//{attribute 'qualified_only'}
{attribute 'strict'}
TYPE E_MotionCommand :
(
	eNoCommand,
	ePower,
	eMoveAbsolute,
	eMoveRelative,
	eMoveVelocity,
	eHalt,
	eGearIn,
	eGearOut
);
END_TYPE

(* stored: Version 1.1.0.1, ProductVersion 3.1.4024.12
   DUT E_MotionCommand: Id {1ca8bf13-8b28-46fc-8a6e-c4e6672e5261} *)
